// TwinCAT 3 PLC project MAIN
// ProgramVersion: 3.1.4026.20
// CompilerDefines: VISU_USEPROPERTYINFO
// libraries:
//   Tc2_Standard, * (Beckhoff Automation GmbH)
//   Tc2_System, * (Beckhoff Automation GmbH)
//   VisuSymbols, 4.5.0.0 (System)
// project tree:
//   / GlobalTextList.TcGTLO, PlcTask.TcTTO, Visualization Manager.TcVMO (not stored)
//   GVLs/ GVL.TcGVL
//   POUs/ FB_SortingMachine.TcPOU, MAIN.TcPOU
//   POUs/Function_block/ E_Color.TcDUT, FB_BaseDiverter.TcPOU, FB_BlueDiverter.TcPOU, FB_YellowDiverter.TcPOU, FB_ColorSensor.TcPOU, FB_Conveyor.TcPOU, FB_RedDiverter.TcPOU, FB_RejectDiverter.TcPOU
//   POUs/Interface/ I_Actuator.TcIO, I_Device.TcIO
//   VISUs/ Visualization.TcVIS
// real-time tasks:
//   TASK PlcTask: cycle T#10ms, priority 20, ADS port 350

CONFIGURATION MAIN
    RESOURCE PLC ON TwinCAT3
        TASK PlcTask(INTERVAL := T#10ms, PRIORITY := 20);
        PROGRAM MAIN WITH PlcTask : MAIN;
    END_RESOURCE
END_CONFIGURATION

// ---- POUs/Function_block/E_Color.TcDUT
TYPE E_Color :
(
    NONE := 0,
    RED := 1,
    BLUE := 2,
	YELLOW := 3,
    UNKNOWN := 4
);
END_TYPE

// ---- GVLs/GVL.TcGVL
{attribute 'qualified_only'}
VAR_GLOBAL

    (* color inputs for each machine *)
    colorMachine : ARRAY[1..10] OF INT;

END_VAR

// ---- POUs/Interface/I_Actuator.TcIO
INTERFACE I_Actuator EXTENDS I_Device

METHOD Start : bool
VAR_INPUT
END_VAR
END_METHOD

METHOD Stop : bool
VAR_INPUT
END_VAR
END_METHOD

END_INTERFACE

// ---- POUs/Interface/I_Device.TcIO

INTERFACE I_Device

METHOD Disable : bool
VAR_INPUT
END_VAR
END_METHOD

METHOD Enable : bool
VAR_INPUT
END_VAR
END_METHOD

METHOD Init : bool
VAR_INPUT
END_VAR
END_METHOD

METHOD Update : bool
VAR_INPUT
END_VAR
END_METHOD

END_INTERFACE

// ---- POUs/MAIN.TcPOU
PROGRAM MAIN
VAR
    machine1 : FB_SortingMachine;
    machine2 : FB_SortingMachine;
    machine3 : FB_SortingMachine;
END_VAR

machine1(machineID := 1);
machine2(machineID := 2);
machine3(machineID := 3);

END_PROGRAM

// ---- POUs/FB_SortingMachine.TcPOU
FUNCTION_BLOCK FB_SortingMachine

VAR_INPUT
    machineID : INT;
END_VAR

VAR
    (* Machine Components *)
    conveyor        : FB_Conveyor;
    sensor : FB_ColorSensor;
    currentColor : E_Color;
	
    redDiverter     : FB_RedDiverter;
    blueDiverter    : FB_BlueDiverter;
	yellowDiverter    : FB_YellowDiverter;
    rejectDiverter  : FB_RejectDiverter;

    (* Machine Status *)
    bInitialized : BOOL ;
    bEnabled     : BOOL;
	bDisabled    : BOOL;

    (* Loop Index *)
    i : INT;

END_VAR

sensor(sensorID := machineID);

currentColor := sensor.GetColor();


(* Sorting decision *)
CASE currentColor OF

    E_Color.RED:
        redDiverter.Start();
		blueDiverter.Stop();
		yellowDiverter.Stop();
		rejectDiverter.Stop();
    E_Color.BLUE:
        blueDiverter.Start();
		redDiverter.Stop();
		yellowDiverter.STop();
		rejectDiverter.Stop();
	E_Color.YELLOW:
		yellowDiverter.Start();
		blueDiverter.Stop();
		redDiverter.Stop();
		rejectDiverter.Stop();
    ELSE
        rejectDiverter.Start();
		redDiverter.Stop();
		blueDiverter.Stop();
		yellowDiverter.Stop();
END_CASE


(* Conveyor always running *)
conveyor.Start();

END_FUNCTION_BLOCK

// ---- POUs/Function_block/FB_Conveyor.TcPOU
FUNCTION_BLOCK FB_Conveyor IMPLEMENTS I_actuator
VAR
    bEnabled : BOOL;
    bRunning : BOOL;
	bDisabled : BOOL;
END_VAR

METHOD Disable : bool
VAR_INPUT
END_VAR
bDisabled := true;
END_METHOD

METHOD Enable : bool
VAR_INPUT
END_VAR
bEnabled := TRUE;
END_METHOD

METHOD Init : bool
VAR_INPUT
END_VAR
bEnabled := FALSE;
bRunning := FALSE;
END_METHOD

METHOD Start : bool
VAR_INPUT
END_VAR
IF bEnabled THEN
    bRunning := TRUE;
	bDisabled := FALSE;
END_IF
END_METHOD

METHOD Stop : bool
VAR_INPUT
END_VAR
IF bDisabled THEN 
	bRunning := FALSE;
	bEnabled := FALSE;
END_IF;
END_METHOD

METHOD Update : bool
VAR_INPUT
END_VAR
IF NOT bEnabled THEN
    bRunning := FALSE;
END_IF
END_METHOD

END_FUNCTION_BLOCK

// ---- POUs/Function_block/FB_ColorSensor.TcPOU
FUNCTION_BLOCK FB_ColorSensor

VAR_INPUT
    sensorID : INT;
END_VAR

VAR
    _color : E_Color := E_Color.UNKNOWN;
    rawColor : INT;
END_VAR

METHOD PUBLIC GetColor : E_Color
VAR
    colorValue : INT;
END_VAR
(* read color from global array *)
rawColor := GVL.colorMachine[sensorID];

CASE rawColor OF
    1: _color := E_Color.RED;
    2: _color := E_Color.BLUE;
    3: _color := E_Color.YELLOW;
ELSE
    _color := E_Color.UNKNOWN;
END_CASE

GetColor := _color;
END_METHOD

METHOD PUBLIC SetColor
VAR_INPUT
    newColor : INT;
END_VAR
IF newColor >= 0 AND newColor <= 4 THEN
    _color := newColor;
END_IF
END_METHOD

END_FUNCTION_BLOCK

// ---- POUs/Function_block/FB_RedDiverter.TcPOU
FUNCTION_BLOCK FB_RedDiverter EXTENDS FB_BaseDiverter
VAR_INPUT
END_VAR
VAR_OUTPUT
END_VAR
VAR
END_VAR

METHOD PUBLIC Sort
VAR_INPUT
    color : E_Color;
END_VAR
IF color = E_Color.RED THEN
    Start();
END_IF
END_METHOD

END_FUNCTION_BLOCK

// ---- POUs/Function_block/FB_BaseDiverter.TcPOU
FUNCTION_BLOCK FB_BaseDiverter IMPLEMENTS I_Actuator
VAR
    bEnabled : BOOL;
    bActive : BOOL;
END_VAR

METHOD Disable : bool
VAR_INPUT
END_VAR
bEnabled := FALSE;
bActive := FALSE;
END_METHOD

METHOD Enable : bool
VAR_INPUT
END_VAR
bEnabled := TRUE;
END_METHOD

METHOD Init : bool
VAR_INPUT
END_VAR
END_METHOD

METHOD Start : bool
VAR_INPUT
END_VAR
IF bEnabled THEN
    bActive := TRUE;
END_IF
END_METHOD

METHOD Stop : bool
VAR_INPUT
END_VAR
bActive := FALSE;
END_METHOD

METHOD Update : bool
VAR_INPUT
END_VAR
END_METHOD

END_FUNCTION_BLOCK

// ---- POUs/Function_block/FB_BlueDiverter.TcPOU
FUNCTION_BLOCK FB_BlueDiverter EXTENDS FB_BaseDiverter
VAR_INPUT
END_VAR
VAR_OUTPUT
END_VAR
VAR
END_VAR

METHOD PUBLIC Sort
VAR_INPUT
    color : E_Color;
END_VAR
IF color = E_Color.BLUE THEN
    Start();
END_IF
END_METHOD

END_FUNCTION_BLOCK

// ---- POUs/Function_block/FB_YellowDiverter.TcPOU
FUNCTION_BLOCK FB_YellowDiverter EXTENDS FB_BaseDiverter
VAR_INPUT
END_VAR
VAR_OUTPUT
END_VAR
VAR
END_VAR

METHOD PUBLIC Sort
VAR_INPUT
    color : E_Color;
END_VAR
IF color = E_Color.YELLOW THEN
    Start();
END_IF
END_METHOD

END_FUNCTION_BLOCK

// ---- POUs/Function_block/FB_RejectDiverter.TcPOU
FUNCTION_BLOCK FB_RejectDiverter EXTENDS FB_BaseDiverter
VAR_INPUT
END_VAR
VAR_OUTPUT
END_VAR
VAR
END_VAR

METHOD PUBLIC Sort
VAR_INPUT
    color : E_Color;
END_VAR
IF color = E_Color.UNKNOWN THEN
    Start();
END_IF
END_METHOD

END_FUNCTION_BLOCK

// ---- GlobalTextList.TcGTLO
TEXTLIST GlobalTextList
  861 = 'Color Detected'
  231 = 'Machine 1'
  18 = 'Machine 2'
  485 = 'Machine 3'
END_TEXTLIST

// ---- VISUs/Visualization.TcVIS
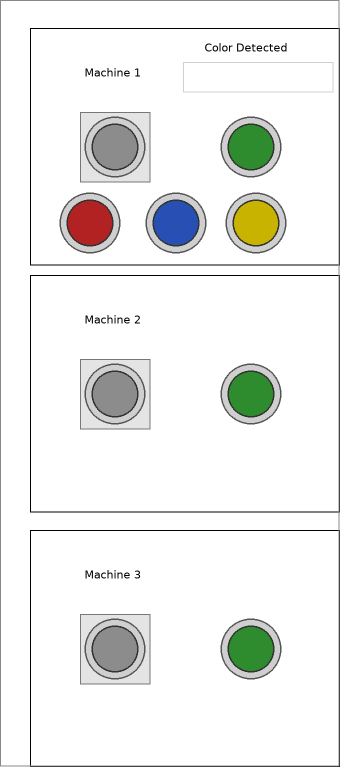
VISUALIZATION Visualization  // 340x767
    Rectangle (30,28 310x237)
    Lamp1 (216,112 70x70), variable: MAIN.machine1.conveyor.bRunning, style: Lamp-Lamp1-Green
    Label (36,44 154x58), "Machine 1"
    PushSwitch (80,112 70x70), variable: MAIN.machine1.conveyor.bRunning, behaviour: TOGGLE, style: Switch-PushSwitch-Gray
    Rectangle (30,275 310x237)
    Lamp1 (216,359 70x70), variable: MAIN.machine2.conveyor.bRunning, style: Lamp-Lamp1-Green
    Label (36,291 154x58), "Machine 2"
    PushSwitch (80,359 70x70), variable: MAIN.machine2.conveyor.bRunning, behaviour: TOGGLE, style: Switch-PushSwitch-Gray
    Rectangle (30,530 310x237)
    Lamp1 (216,614 70x70), variable: MAIN.machine3.conveyor.bRunning, style: Lamp-Lamp1-Green
    Label (36,546 154x58), "Machine 3"
    PushSwitch (80,614 70x70), variable: MAIN.machine3.conveyor.bRunning, behaviour: TOGGLE, style: Switch-PushSwitch-Gray
    Textfield (183,62 150x30), text variable: MAIN.machine1.currentColor
    Lamp1 (55,188 70x70), variable: MAIN.machine1.redDiverter.bActive, style: Lamp-Lamp1-Red
    Lamp1 (141,188 70x70), variable: MAIN.machine1.blueDiverter.bActive, style: Lamp-Lamp1-Blue
    Lamp1 (221,188 70x70), variable: MAIN.machine1.yellowDiverter.bActive, style: Lamp-Lamp1-Yellow
    Label (169,19 154x58), "Color Detected"
END_VISUALIZATION
